% RSLogix 500 project PID SUBSTITUTION_BAK009.RSS, saved by version 8.30.00.16 %
PROJECT "UNTITLED"    % processor: Bul.1763 MicroLogix 1100 Series B %

PROGRAM FILES
  LAD 2 "MAIN"  8 rungs

DATA FILES
  O0 OUTPUT  4 elements
  I1 INPUT  6 elements
  S2 STATUS  66 elements
  B3 BINARY  1 elements
  T4 TIMER  1 elements
  C5 COUNTER  1 elements
  R6 CONTROL  1 elements
  N7 INTEGER  20 elements
  F8 FLOAT  1 elements

LADDER 2 "MAIN"
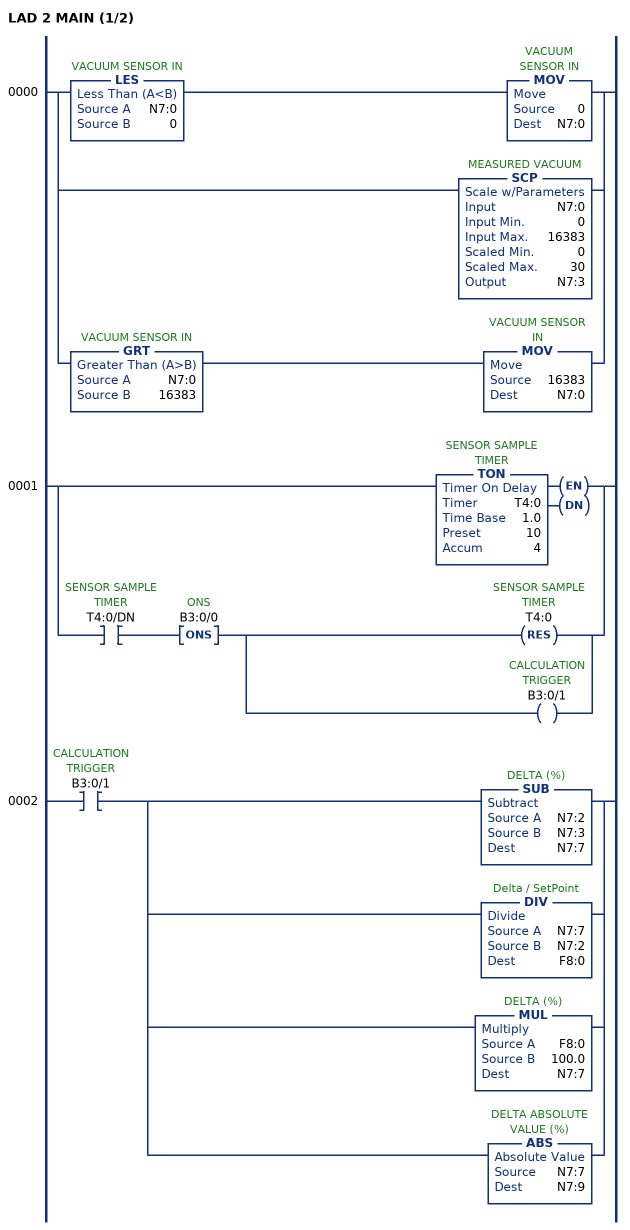
% Rung: 0 %
SOR BST LES N7:0 0 MOV 0 N7:0 NXB SCP N7:0 0 16383 0 30 N7:3 NXB GRT N7:0 16383 MOV 16383 N7:0 BND EOR
%   N7:0  "VACUUM SENSOR IN" %
%   N7:3  "MEASURED VACUUM" %
% Rung: 1 %
SOR BST TON T4:0 1.0 10 4 NXB XIC T4:0/DN ONS B3:0/0 BST RES T4:0 NXB OTE B3:0/1 BND BND EOR
%   T4:0  "SENSOR SAMPLE TIMER" %
%   B3:0/0  "ONS" %
%   B3:0/1  "CALCULATION TRIGGER" %
% Rung: 2 %
SOR XIC B3:0/1 BST SUB N7:2 N7:3 N7:7 NXB DIV N7:7 N7:2 F8:0 NXB MUL F8:0 100.0 N7:7 NXB ABS N7:7 N7:9 BND EOR
%   B3:0/1  "CALCULATION TRIGGER" %
%   N7:2  "VACUM SETPOINT" %
%   N7:3  "MEASURED VACUUM" %
%   N7:7  "DELTA (%)" %
%   F8:0  "Delta / SetPoint" %
%   N7:9  "DELTA ABSOLUTE VALUE (%)" %

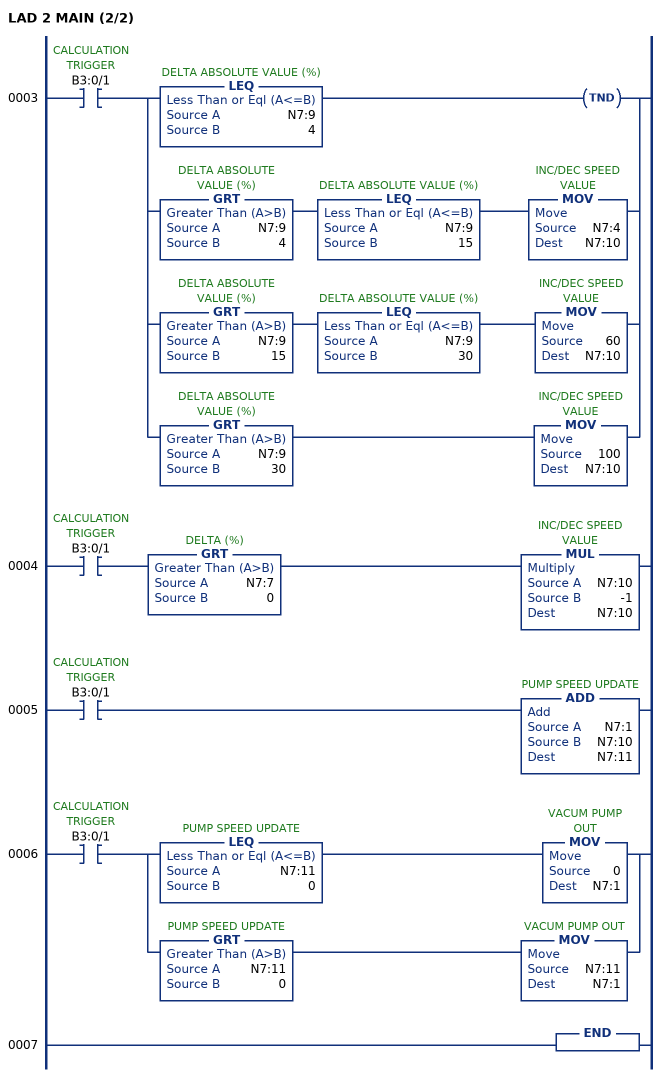
% Rung: 3 %
SOR XIC B3:0/1 BST LEQ N7:9 4 TND NXB GRT N7:9 4 LEQ N7:9 15 MOV N7:4 N7:10 NXB GRT N7:9 15 LEQ N7:9 30 MOV 60 N7:10 NXB GRT N7:9 30 MOV 100 N7:10 BND EOR
%   B3:0/1  "CALCULATION TRIGGER" %
%   N7:9  "DELTA ABSOLUTE VALUE (%)" %
%   N7:4  "SPEED INC/DEC 4-15%" %
%   N7:10  "INC/DEC SPEED VALUE" %
% Rung: 4 %
SOR XIC B3:0/1 GRT N7:7 0 MUL N7:10 -1 N7:10 EOR
%   B3:0/1  "CALCULATION TRIGGER" %
%   N7:7  "DELTA (%)" %
%   N7:10  "INC/DEC SPEED VALUE" %
% Rung: 5 %
SOR XIC B3:0/1 ADD N7:1 N7:10 N7:11 EOR
%   B3:0/1  "CALCULATION TRIGGER" %
%   N7:1  "VACUM PUMP OUT" %
%   N7:10  "INC/DEC SPEED VALUE" %
%   N7:11  "PUMP SPEED UPDATE" %
% Rung: 6 %
SOR XIC B3:0/1 BST LEQ N7:11 0 MOV 0 N7:1 NXB GRT N7:11 0 MOV N7:11 N7:1 BND EOR
%   B3:0/1  "CALCULATION TRIGGER" %
%   N7:11  "PUMP SPEED UPDATE" %
%   N7:1  "VACUM PUMP OUT" %
% Rung: 7 %
SOR END EOR

OTHER DOCUMENTED ADDRESSES
  N7:5  "SPEED INC/DEC 15-30%"
  N7:6  "SPEED INC/DEC >30%"
  N7:8  "ABSOLUT VALUE OF DELTA ABS(DELTA)"

DATA TABLE (non-zero values as saved)
DATA T4
% .PRE .ACC %
% T4:0 % 10 4
DATA N7
% N7:0 % 8192 6000 15 0 20 60 100 0 0 0
